IF iState >= 10 AND iState < 100 THEN 
	THIS^.M_0ReadActConfig();
ELSIF iState >= 1000 AND iState < 1100 THEN
//	act11_DownloadDriveFirmware();				// Execute this Action in a different Task
 	iState := 100; 
ELSIF iState >= 100 AND iState < 200 THEN
	THIS^.M_1ConfigAxes();
ELSIF iState >= 200 AND iState < 300 THEN
	THIS^.M_2ConfigSercosIO();
ELSIF iState >= 300 AND iState < 400 THEN
	THIS^.M_3ConfigInlineIO();	
ELSIF iState >= 400 AND iState < 500 THEN
	THIS^.M_4ConfigProfibsIO();
ELSIF iState >= 500 AND iState < 600 THEN
	iState := 800;
ELSIF iState >= 800 AND iState < 900 THEN
	THIS^.M_8WriteConfig();
ELSIF iState >= 900 AND iState < 1000 THEN
	THIS^.M_9ErrorDone();
END_IF
END_METHOD

METHOD PRIVATE M_GetSafetyType : STRING(2)
VAR_INPUT
	///Temp string to prepare elements;
	apsTypeCodeElements: ARRAY[1..20] OF POINTER TO STRING(255);
	bSecondDoubleAxis: BOOL := FALSE;
END_VAR
IF (LEFT (apsTypeCodeElements[1]^,5) = 'CSH01') THEN

	M_GetSafetyType := apsTypeCodeElements[6]^;
	
ELSIF	(LEFT (apsTypeCodeElements[1]^,5) = 'CDB01') THEN

	M_GetSafetyType := apsTypeCodeElements[7]^;
	
ELSIF	(LEFT (apsTypeCodeElements[1]^,5) = 'CSE02') 
OR	(LEFT (apsTypeCodeElements[1]^,5) = 'CSB02')
OR	(LEFT (apsTypeCodeElements[1]^,5) = 'CSH02') 
OR	(LEFT (apsTypeCodeElements[1]^,5) = 'CSB01') 
OR	(LEFT (apsTypeCodeElements[1]^,5) = 'KMC02') THEN		(* 2019-03-21 Bär: Typ 'KMC02' im Rahmen der RDK90 (Mi-Antriebe) hinzugefügt *)

	M_GetSafetyType := apsTypeCodeElements[5]^;
	
ELSIF	(LEFT (apsTypeCodeElements[1]^,5) = 'CDB02') THEN

	IF NOT bSecondDoubleAxis THEN
		M_GetSafetyType := apsTypeCodeElements[6]^;
	ELSE	
		M_GetSafetyType := apsTypeCodeElements[7]^;
	END_IF
	
ELSIF	(LEFT (apsTypeCodeElements[1]^,5) = 'HCS01') THEN

	M_GetSafetyType := apsTypeCodeElements[9]^;
	
ELSIF	(LEFT (apsTypeCodeElements[1]^,5) = 'KSM02') 
OR	(LEFT (apsTypeCodeElements[1]^,5) = 'KMS02')THEN

	M_GetSafetyType := apsTypeCodeElements[7]^;
	
END_IF
END_METHOD

///FUNCTION FUN_GetSercosAdress
///
///General Header
///----------------------------------------------------------------------------------------------
///Short description      : extract sercos adress for double axis config
///Version                : 13.0.0
///Author                 : Jörg Schneider
///Date                   : 13-07-12 15:46:38
///Company                : DC-IA
///Target                 : MLC 13 ff
///----------------------------------------------------------------------------------------------
METHOD PRIVATE M_GetSercosAdress : INT
VAR_INPUT
	/// Pointer to String Element of C-0-0479 e.g. 'V3|34' 
	pbToElement: POINTER TO BYTE;
	/// First or second Adress of doubleAxis
	iNoOfAddress: INT;
END_VAR
VAR
	sTemp: STRING := '';
	sTemp2: STRING := '';
	pbTemp: POINTER TO BYTE;
	pbTemp2: POINTER TO BYTE;
	psStringTemp: POINTER TO STRING(1);
	bTemp: BYTE;
	iDigit1: INT;
	iDigit2: INT;
END_VAR
// copy first sign to stTemp 				
pbTemp := pbToElement+1;	
psStringTemp := pbTemp;					
sTemp := psStringTemp^;
bTemp := pbTemp^;
		
sTemp2 := '';		
pbTemp2 := ADR (sTemp2);



// Do until '|' or end of string appears				
IF NOT (sTemp = '') 			// End of String
AND NOT (bTemp = 124) THEN		// Or '|' character
	pbTemp2^:= pbTemp^;

	iDigit1 := STRING_TO_INT(sTemp);
	iDigit2 := 0;
	
	pbTemp := pbTemp + 1;
	pbTemp2 := pbTemp2 + 1;
	psStringTemp := pbTemp;
	sTemp := psStringTemp^;
	bTemp := pbTemp^;

	
END_IF	

IF NOT (sTemp = '') 
AND NOT (bTemp = 124) THEN
	pbTemp2^:= pbTemp^;
	
	iDigit1 := iDigit1 *10;
	iDigit2 := STRING_TO_INT(sTemp);
		
	pbTemp := pbTemp + 1;
	pbTemp2 := pbTemp2 + 1;
	psStringTemp := pbTemp;
	sTemp := psStringTemp^;
	bTemp := pbTemp^;
	
END_IF	


IF iNoOfAddress = 2 THEN 
	//Reset Temp variable
	sTemp2 := '';		
	pbTemp2 := ADR (sTemp2);
	pbTemp := pbTemp + 1;
	psStringTemp := pbTemp;
	sTemp := psStringTemp^;


	IF NOT (sTemp = '')  THEN
		pbTemp2^:= pbTemp^;
					
		iDigit1 := STRING_TO_INT(sTemp);
		iDigit2 := 0;
				
		pbTemp := pbTemp + 1;
		pbTemp2 := pbTemp2 + 1;
		psStringTemp := pbTemp;
		sTemp := psStringTemp^;
		bTemp := pbTemp^;
	
	END_IF	
	
	IF NOT (sTemp = '')  THEN
		pbTemp2^:= pbTemp^;
		
		iDigit1 := iDigit1 *10;
		iDigit2 := STRING_TO_INT(sTemp);
		
		pbTemp := pbTemp + 1;
		pbTemp2 := pbTemp2 + 1;
		psStringTemp := pbTemp;
		sTemp := psStringTemp^;
		bTemp := pbTemp^;
		
		
	END_IF	

END_IF


M_GetSercosAdress := iDigit1 + iDigit2;
END_METHOD

METHOD PRIVATE M_S20TypeToString : STRING
VAR_INPUT
	eS20Type: E_S20Type;
END_VAR
CASE eS20Type OF
	
	E_S20Type.S20_UNDEFINED				:	M_S20TypeToString :=  'undefinded'				;
	E_S20Type.S20_S3_BK_PLUS				:	M_S20TypeToString :=  'S20-S3-BK+'	            ;
	E_S20Type.S20_DI_16_4     		   	:	M_S20TypeToString :=  'S20-DI-16/4'	            ;
	E_S20Type.S20_DO_16_3          		:	M_S20TypeToString :=  'S20-DO-16/3'	            ;
	E_S20Type.S20_DI_32_1          		:	M_S20TypeToString :=  'S20-DI-32/1'	            ;
	E_S20Type.S20_DO_32_1          		:	M_S20TypeToString :=  'S20-DO-32/1'	            ;
	E_S20Type.S20_DO_8_2_2A        		:	M_S20TypeToString :=  'S20-DO-8/2-2A'            ;
	E_S20Type.S20_DI_16_1          		:	M_S20TypeToString :=  'S20-DI-16/1'	            ;
	E_S20Type.S20_DO_16_1          		:	M_S20TypeToString :=  'S20-DO-16/1'	            ;
	E_S20Type.S20_AI_8             		:	M_S20TypeToString :=  'S20-AI-8'		            ;
	E_S20Type.S20_AI_8_RTD         		:	M_S20TypeToString :=  'S20-AI-8-RTD'	            ;
	E_S20Type.S20_AI_8_UTH         		:	M_S20TypeToString :=  'S20-AI-8-UTH'	            ;
	E_S20Type.S20_AO_8             		:	M_S20TypeToString :=  'S20-AO-8'		            ;
	E_S20Type.S20_CNT_INC_2_2      		:	M_S20TypeToString :=  'S20-CNT-INC-2/2'	        ;
	E_S20Type.S20_SSI_AO_1_1       		:	M_S20TypeToString :=  'S20-SSI-AO-1/1'	        ;
	E_S20Type.Placeholder_1          		:	M_S20TypeToString :=  'Test_ChM'			        ;
	E_S20Type.Placeholder_2 		     	:	M_S20TypeToString :=  'Test_ChM'			        ;
	E_S20Type.Placeholder_3          		:	M_S20TypeToString :=  'Test_ChM'			        ;
	E_S20Type.S20_AI_4_I           		:	M_S20TypeToString :=  'S20-AI-4-I'		        ;
	E_S20Type.S20_AI_4_U           		:	M_S20TypeToString :=  'S20-AI-4-U'		        ;
	E_S20Type.S20_DI_64_1    			   	:	M_S20TypeToString :=  'S20-DI-64/1'		        ;
	E_S20Type.S20_DI_16_1_HS     	 		:	M_S20TypeToString :=  'S20-DI-16/1-HS'	        ;
	E_S20Type.S20_AI_4_RTD         		:	M_S20TypeToString :=  'S20-AI-4-RTD'		        ;
	E_S20Type.S20_RS_UNI           		:	M_S20TypeToString :=  'S20-RS-UNI'		        ;
	E_S20Type.S20_DIDO_8_1         		:	M_S20TypeToString :=  'S20-DIDO-8/1'		        ;
	E_S20Type.S20_AO_4             		:	M_S20TypeToString :=  'S20-AO-4'                 ;
	E_S20Type.S20_AI_4_UTH         		:	M_S20TypeToString :=  'S20-AI-4-UTH'		        ;
	E_S20Type.S20_SSDI_8_4               	:	M_S20TypeToString:=  'SSDI-8/4'			        ;
	E_S20Type.S20_SSDO_8_3               	:	M_S20TypeToString:=  'SSDO-8/3'			        ;
	E_S20Type.S20_AI6_AO2_SSI2     		:	M_S20TypeToString:=  'S20-AI6-AO2-SSI2'	        ;
	E_S20Type.S20_INC_2            		:	M_S20TypeToString:=  'S20-INC-2'		        ;
	E_S20Type.S20_AIAO_2           		:	M_S20TypeToString:=  'S20-AIAO-2'		        ;
	E_S20Type.S20_DO_64_1          		:	M_S20TypeToString:=  'S20-DO-64/1'				;	
	E_S20Type.S20_DOR_4_2_220_AC   		:	M_S20TypeToString:=  'S20-DOR-4/2-220-AC'		;	
	E_S20Type.S20_DI_16_4_DO_8_3_HS		:	M_S20TypeToString:=  'S20-DI-16/4-DO-8/3-HS'	;	
															  	
END_CASE
END_METHOD

METHOD PRIVATE M_TypeCodeIsRexrothIO : BOOL
VAR_INPUT
	sTypeCode: STRING;
END_VAR

IF sTypeCode = 'L05R911172531' THEN			// S20-S3-BK
	M_TypeCodeIsRexrothIO := TRUE;
ELSIF 	sTypeCode = 'L05R911173318' THEN		// S20-S3-BK+
	M_TypeCodeIsRexrothIO := TRUE;
ELSIF 	sTypeCode = 'L05R911170875' THEN		// R-IL S3 BK DI8 DO4-PAC
	M_TypeCodeIsRexrothIO := TRUE;	
ELSIF 	sTypeCode = 'L05R911170874' THEN		// R-ILB S3 AI4 AO2
	M_TypeCodeIsRexrothIO := TRUE;
ELSIF 	sTypeCode = 'L05R911171676' THEN		// R-ILB S3 AI6 AO4/F
	M_TypeCodeIsRexrothIO := TRUE;
ELSIF 	sTypeCode = 'L05R911171949' THEN		// R-ILB S3 AI12 AO4 SSI-IN4
	M_TypeCodeIsRexrothIO := TRUE;
ELSIF 	sTypeCode = 'L05R911170826' THEN		// R-ILB S3 24 DI16 DIO16
	M_TypeCodeIsRexrothIO := TRUE;
ELSIF 	sTypeCode = 'L05R911171675' THEN		// R-ILB S3 24 DI16 DIO16/F
	M_TypeCodeIsRexrothIO := TRUE;
ELSIF 	sTypeCode = 'L05R911172899' THEN		// S67-S3-BK-DI8-M8
	M_TypeCodeIsRexrothIO := TRUE;

ELSE 	
	M_TypeCodeIsRexrothIO := FALSE;
END_IF
END_METHOD

END_FUNCTION_BLOCK

// GeneralFunctionBlocks/ActivateDevices/ITF_ActivateDevices
INTERFACE ITF_ActivateDevices

METHOD M_Execute
END_METHOD

END_INTERFACE

// GeneralFunctionBlocks/ChangeNextDiagDelay/FB_ChangeNextDiagDelay
{attribute 'qualified_only' := ''}
{attribute 'namespace' := 'ILGStdLib.FunctionBlocks'}
FUNCTION_BLOCK FB_ChangeNextDiagDelay
VAR_INPUT
	/// start procedure
	IN_bExecute: BOOL;
	/// Delay Time in ms
	IN_diDiagDelayTime: DINT;
END_VAR
VAR_OUTPUT
	/// Done
	OUT_bDone: BOOL;
	/// Active
	OUT_bActive: BOOL;
	/// error	
	OUT_bError: BOOL;
	/// internat state when error occured
	OUT_iErrorState: INT;
END_VAR
VAR CONSTANT
	/// max no of directory entries
	iMaxDirEntry: INT := 400;
END_VAR
VAR
	bExecuteOld: BOOL;
	istate: INT;
	iLength: INT;
	i: INT;
	j: INT;
	iEOF: INT;
	hCfg: ITF_FILEASYNC;
	sBuffer: STRING(7000);
	udiReadBytes: UDINT;
	udiFileSize: UDINT;
	sLineFeed: STRING(1);
	sTemp: STRING;
	sTemp2: STRING;
	sSearch: STRING;
	diResult: DINT;
	astSplit: ST_Split;
	asStringFile: ARRAY[1..iMaxDirEntry] OF STRING;
	psFileName : POINTER TO STRING;
	psNewFileName : POINTER TO STRING;
	fb_ILFileDeleteAsync: IL_FileDeleteAsync;
	fb_ILFileOpenAsync: IL_FileAsync;
	fb_ILFileReadAsync: IL_FileReadAsync;	
	fb_ILFileGetSizeAsync: IL_FileGetSizeAsync;
	fb_ILFileRenameAsync: IL_FileRenameAsync;
	fb_ILFileWriteAsync: IL_FileWriteAsync;
END_VAR


IF IN_bExecute AND NOT bExecuteOld THEN
	bExecuteOld := TRUE;
	OUT_bActive := TRUE;
	OUT_bDone := FALSE;
	OUT_bError := FALSE;
	iState := 40;
END_IF	

IF NOT IN_bExecute AND bExecuteOld 
	AND (OUT_bDone OR OUT_bError) THEN
	bExecuteOld := FALSE;
	OUT_bActive := FALSE;
	OUT_bDone := FALSE;
	OUT_bError := FALSE;
	iState := 0;
END_IF	


CASE istate OF

40: // Größe ermitteln
	psFileName^:= '/ata0a/ProjectData/PLC/DevicePLcAdd.cfg';
	OUT_iErrorState := iState;
	fb_ILFileGetSizeAsync(
		Execute:=TRUE , 
		FileName:= psFileName,			(* 2016-10 gt: IW13: '/ata0a/DevicePLcAdd.cfg' --> IW14: '/ata0a/ProjectData/PLC/DevicePLcAdd.cfg' *) (* 2017-01-26 gt: relevant für IW14 *)
		Done=> ,		
		Active=> ,
		Error=> ,
 		ErrorId=> ,
		ErrorIdent=> , 
		FileSize=> udiFileSize);

	IF fb_ILFileGetSizeAsync.Done THEN
		fb_ILFileGetSizeAsync(
			Execute:= FALSE);
		iState :=50;
	END_IF
	// Error	
	IF fb_ILFileGetSizeAsync.Error THEN
		fb_ILFileGetSizeAsync(
			Execute:= FALSE);
		iState :=999;
	END_IF
			
50:	// DevicePlcAdd.cfg öffnen
	psFileName^:= '/ata0a/ProjectData/PLC/DevicePLcAdd.cfg';
	OUT_iErrorState := iState;		
	fb_ILFileOpenAsync(
		Enable:= TRUE, 
		FileName:=psFileName,		(* 2016-10 gt: IW13: '/ata0a/DevicePLcAdd.cfg' --> IW14: '/ata0a/ProjectData/PLC/DevicePLcAdd.cfg' *) (* 2017-01-26 gt: relevant für IW14 *)
		Mode:=  AM_READ,
		InOperation=> , 
		Active=> ,
		Shutdown=> , 		 
		Error=> , 
		ErrorId=> ,
		ErrorIdent=> , 
		FileHandle=> hCfg);

	IF fb_ILFileOpenAsync.InOperation THEN		
		sBuffer := '';	
		iState :=60;
	END_IF

	// Error	
	IF fb_ILFileOpenAsync.Error THEN
		fb_ILFileOpenAsync(
			Enable:= FALSE);
		iState :=999;
	END_IF
		
60:	// DevicePlcAdd.cfg lesen
	OUT_iErrorState := iState;
	fb_ILFileReadAsync(
		Execute:= TRUE,
		BufferAddr:= ADR(sBuffer),
 		BufferSize:= udiFileSize, 
		FileHandle:= hCfg,  
		Done=> , 
		Active=> , 
		Error=> , 
		ErrorId=> ,
		ErrorIdent=> , 
		BytesRead=> udiReadBytes );

	IF fb_ILFileReadAsync.Done THEN
		fb_ILFileReadAsync(
			Execute:= FALSE);
		iState := 70;
	END_IF

	// Error	
	IF fb_ILFileReadAsync.Error THEN
		fb_ILFileReadAsync(
			Execute:= FALSE);
		iState :=999;
	END_IF
	
70: // Datei schließen
	OUT_iErrorState := iState;
	fb_ILFileOpenAsync(
		Enable:= FALSE); 

	IF (fb_ILFileOpenAsync.InOperation = FALSE) THEN
		iState :=80;
	END_IF

	// Error	
	IF fb_ILFileOpenAsync.Error THEN
		iState :=999;
	END_IF
	
	(* Auskommentiert, da strSplit strLen usw. noch fehlen
80: // Datei in Array of String kopieren und Formatzeichen löschen
	OUT_iErrorState := iState;
	strSplit(ADR(sBuffer),13 ,0,FALSE,ADR(astSplit));
	sLineFeed := CHR(10);
	
	FOR i := 1 TO iMaxDirEntry DO 
		IF astSplit.arWords[i]^ = astSplit.arWords[iMaxDirEntry]^ THEN 
			iEOF := i ;		
			i := iMaxDirEntry;
		END_IF
		asStringFile[i] := DEL_CHARS(astSplit.arWords[i]^, sLineFeed);
	END_FOR
	
	// letzte Zeile löschen
	asStringFile[iEOF-1] := ''; 
	iEOF	:= iEOF-2;
	
	iState := 90;	

90:	// Sektion im File suchen
	OUT_iErrorState := iState;
	sSearch := '[NetX_Device]';  
	iLength :=	strLen(ADR(sSearch));
	FOR i := 1 TO iEOF DO
		sTemp := '';
		IF strLen(ADR(asStringFile[i])) >= iLength THEN									// Text länger als strSearch
			
			IF (asStringFile[i] = sSearch) THEN					// Text enthält '[NetX_Device]'
				sSearch := 'NetxDiagDelayTime=';
				iLength :=	strLen(ADR(sSearch));
				strNCopy(ADR(sTemp), (INT_TO_UINT(iLength)+2), ADR(asStringFile[i+1]), iLength);		(* 2014-11-14 gt: INT_TO_UINT() hinzu, wegen Warnung *)
				
				IF NOT (sTemp = sSearch) THEN					// Text enthält noch nicht 'NetxDiagDelayTime='
					FOR j:= iEOF TO i+1 BY -1 DO					// dann alle Zeilen um eins nach unten verschieben
						asStringFile[j+1] := asStringFile[j];	
					END_FOR
			
					asStringFile[i+1] := 'NetxDiagDelayTime=';		// Zeile inzufügen.
					sTemp := DINT_TO_STRING(IN_diDiagDelayTime);
					strConcat(ADR(asStringFile[i+1]), SIZEOF(asStringFile[i+1]), ADR(sTemp));
				ELSE																	// Text enthält 'NetxDiagDelayTime='
					sTemp := 'NetxDiagDelayTime=';		
					sTemp2 := DINT_TO_STRING(IN_diDiagDelayTime);
					strConcat(ADR(sTemp), SIZEOF(sTemp), ADR(sTemp2));
					IF sTemp = asStringFile[i+1] THEN  // Vergleichen, ob Wert stimmt 
						i := iEOF+1;
						iState := 250;  									// --> Done
						RETURN;
					ELSE
						asStringFile[i+1] := sTemp; 		// Zeile neu schreiben
					END_IF		
				END_IF
				i := iEOF+1; // End FOR Loop
			END_IF
		END_IF	
	END_FOR	
	
	iState := 110;
	*)
110: // DevicePlcAdd.new neu anlegen und zum schreiben öffnen
	psFileName^:= '/ata0a/ProjectData/PLC/DevicePLcAdd.new';
	OUT_iErrorState := iState;
	// hCfg := SysFileStreamFOpenV3('/ata0a/ProjectData/PLC/DevicePLcAdd.new', 'w');		(* 2016-10 gt: IW13: ('/ata0a/DevicePLcAdd.new', 'w') --> IW14: ('/ata0a/ProjectData/PLC/DevicePLcAdd.new', 'w') *)	(* 2017-01-26 gt: relevant für IW14 *)
	fb_ILFileOpenAsync(
		Enable:= TRUE, 
		FileName:=psFileName,		(* 2016-10 gt: IW13: '/ata0a/DevicePLcAdd.cfg' --> IW14: '/ata0a/ProjectData/PLC/DevicePLcAdd.cfg' *) (* 2017-01-26 gt: relevant für IW14 *)
		Mode:=  AM_WRITE,
		InOperation=> , 
		Active=> ,
		Shutdown=> , 		 
		Error=> , 
		ErrorId=> ,
		ErrorIdent=> , 
		FileHandle=> hCfg);

	IF fb_ILFileOpenAsync.InOperation THEN					
		iState :=120;
		j := 0;
	END_IF

	// Error	
	IF fb_ILFileOpenAsync.Error THEN
		fb_ILFileOpenAsync(
			Enable:= FALSE);
		iState :=999;
	END_IF
		
	
120:
	OUT_iErrorState := iState;
	FOR i := j+1 TO iEOF DO
		diResult := FUN_WriteLnString(hCfg, asStringFile[i]);
(*		IF i >= j+10 THEN
			j := i;
			RETURN;
		END_IF  	*)
	END_FOR
	iState :=130;

130:
	OUT_iErrorState := iState;
	
	fb_ILFileOpenAsync(
		Enable:= FALSE);
	iState :=140;

140: // alte Datei umbenennen
	psFileName^ := '/ata0a/ProjectData/PLC/DevicePLcAdd.cfg';
	psNewFileName^ := '/ata0a/ProjectData/PLC/DevicePLcAdd.old'; 
	OUT_iErrorState := iState;
	fb_ILFileRenameAsync(
		Execute:= TRUE, 
		OldName:= psFileName, 		(* 2016-10 gt: IW13: '/ata0a/DevicePLcAdd.cfg' --> IW14: '/ata0a/ProjectData/PLC/DevicePLcAdd.cfg' *)	(* 2017-01-26 gt: relevant für IW14 *)
		NewName:= psNewFileName, 		(* 2016-10 gt: IW13: '/ata0a/DevicePLcAdd.old' --> IW14: '/ata0a/ProjectData/PLC/DevicePLcAdd.old' *)	(* 2017-01-26 gt: relevant für IW14 *)
		Done=> , 
		Active=> , 
		Error=> , 
		ErrorId=> ,
		ErrorIdent=>);
	
	IF fb_ILFileRenameAsync.Done THEN
		fb_ILFileRenameAsync(
			Execute:= FALSE);
		iState :=150;
	END_IF

		// Error	
	IF fb_ILFileRenameAsync.Error THEN
		fb_ILFileRenameAsync(
			Execute:= FALSE);
		iState :=999;
	END_IF

150: // neue Datei umbenennen
	psFileName^ := '/ata0a/ProjectData/PLC/DevicePLcAdd.new';
	psNewFileName^ := '/ata0a/ProjectData/PLC/DevicePLcAdd.cfg';
	OUT_iErrorState := iState;	
	fb_ILFileRenameAsync(
		Execute:= TRUE, 
		OldName:= psFileName, 		(* 2016-10 gt: IW13: '/ata0a/DevicePLcAdd.new' --> IW14: '/ata0a/ProjectData/PLC/DevicePLcAdd.new' *)	(* 2017-01-26 gt: relevant für IW14 *)
		NewName:= psNewFileName,		(* 2016-10 gt: IW13: '/ata0a/DevicePLcAdd.cfg' --> IW14: '/ata0a/ProjectData/PLC/DevicePLcAdd.cfg' *) (* 2017-01-26 gt: relevant für IW14 *)
		Done=> , 
		Active=> , 
		Error=> , 
		ErrorId=> ,
		ErrorIdent=> );
	
	IF fb_ILFileRenameAsync.Done THEN
		fb_ILFileRenameAsync(
			Execute:= FALSE);
		iState :=160;
	END_IF

	// Error	
	IF fb_ILFileRenameAsync.Error THEN
		fb_ILFileRenameAsync(
			Execute:= FALSE);
		iState :=999;
	END_IF
	
160: // alte Datei löschen
	psFileName^ := '/ata0a/ProjectData/PLC/DevicePLcAdd.old';
	OUT_iErrorState := iState;
	fb_ILFileDeleteAsync(
		Execute:= TRUE, 
		FileName:= psFileName, 		(* 2016-10 gt: IW13: '/ata0a/DevicePLcAdd.old' --> IW14: '/ata0a/ProjectData/PLC/DevicePLcAdd.old' *)	(* 2017-01-26 gt: relevant für IW14 *)
		Done=> , 
		Active=> , 
		Error=> , 
		ErrorId=> ,
		ErrorIdent=> );
	
	IF fb_ILFileDeleteAsync.Done THEN
		fb_ILFileDeleteAsync(
			Execute:= FALSE);
		i := 0;
		iState :=250;
	END_IF

	// Error	
	IF fb_ILFileDeleteAsync.Error THEN
		fb_ILFileDeleteAsync(
			Execute:= FALSE);
		iState :=999;
	END_IF

250:  // Done
	OUT_iErrorState := 0;
	OUT_bDone := TRUE;
	OUT_bActive := FALSE;	
	OUT_bError := FALSE;

999: // ERROR 
	OUT_bDone := FALSE;
	OUT_bActive := FALSE;	
	OUT_bError := TRUE;
	
END_CASE

END_FUNCTION_BLOCK

// GeneralFunctions/Convert/F_byWordToLeftByte
{attribute 'qualified_only' := ''}
{attribute 'namespace' := 'ILGStdLib.Functions.Convert'}
FUNCTION F_byWordToLeftByte : BYTE
VAR_INPUT
	/// Zu spaltendes Wort 
	In_wInput: WORD;
END_VAR
VAR
	pwWord: POINTER TO WORD;
	wTEMP: WORD;
END_VAR

pwWord:= ADR(In_wInput);
pwWord:= (pwWord+1);
wTEMP:= pwWord^;
F_byWordToLeftByte:= WORD_TO_BYTE(wTEMP);

END_FUNCTION

// GeneralFunctions/Convert/F_DwordToStrH5
{attribute 'qualified_only' := ''}
{attribute 'namespace' := 'ILGStdLib.Functions.Convert'}
FUNCTION F_DwordToStrH5 : STRING(5)
VAR_INPUT
	In_dwInput: DWORD;
END_VAR
VAR
	i: INT;
	byTemp: BYTE;
	pbyOut: POINTER TO BYTE;
END_VAR

//read output adress
pbyOut := ADR(F_DwordToStrH5) + 5;
// write last byte of String 
pbyOut^:= 0;

// write the 5 hex characters backwards 
FOR i := 1 TO 5 DO
	//decrement pointer
	pbyOut := pbyOut - 1;
	// read the lowest value
	byTemp := DWORD_TO_BYTE(In_dwInput AND 16#0000F);
	// convert value to hex 
	IF (byTemp <= 9) THEN 
		byTemp := byTemp + 48; 
	ELSE 
		byTemp := byTemp + 55; 
	END_IF
	// write value to string
	pbyOut^ := byTemp;
	//shift input for next hex digit
	In_dwInput := SHR(In_dwInput,4);
END_FOR

END_FUNCTION

// GeneralFunctions/Convert/F_DwordToStrH8
{attribute 'qualified_only' := ''}
{attribute 'namespace' := 'ILGStdLib.Functions.Convert'}
FUNCTION F_DwordToStrH8 : STRING(8)
VAR_INPUT
	In_dwInput: DWORD;
END_VAR
VAR
	i: INT;
	byTemp: BYTE;
	pbyOut: POINTER TO BYTE;
END_VAR

//read output adress
pbyOut := ADR(F_DwordToStrH8) + 8;
// write last byte of String 
pbyOut^:= 0;

// write the 8 hex characters backwards 
FOR i := 1 TO 8 DO
	//decrement pointer
	pbyOut := pbyOut - 1;
	// read the lowest value
	byTemp := DWORD_TO_BYTE(In_dwInput AND 16#0000000F);
	// convert value to hex 
	IF (byTemp <= 9) THEN 
		byTemp := byTemp + 48; 
	ELSE 
		byTemp := byTemp + 55; 
	END_IF
	// write value to string
	pbyOut^ := byTemp;
	//shift input for next hex digit
	In_dwInput := SHR(In_dwInput,4);
END_FOR

END_FUNCTION

// GeneralFunctions/Convert/F_dwSwapDWordWord
{attribute 'qualified_only' := ''}
{attribute 'namespace' := 'ILGStdLib.Functions.Convert'}
FUNCTION F_dwSwapDWordWord : DWORD
VAR_INPUT
	In_dwInput: DWORD;
END_VAR
VAR
	pwWordIn: POINTER TO ARRAY[1..2] OF WORD;
	pwWordOut: POINTER TO ARRAY[1..2] OF WORD;
	dwOutput: DWORD;
END_VAR


pwWordIn := ADR(In_dwInput);
pwWordOut := ADR(dwOutput);

pwWordOut^[1]	:=	pwWordIn^[2] ;
pwWordOut^[2]	:=	pwWordIn^[1] ;

F_dwSwapDWordWord := dwOutput;

END_FUNCTION

// GeneralFunctions/Convert/F_iAnalogOutput4To20mA
{attribute 'qualified_only' := ''}
{attribute 'namespace' := 'ILGStdLib.Functions.Convert'}
FUNCTION F_iAnalogOutput4To20mA : INT
VAR_INPUT
	/// x;  Wert zur Wandlung für die Analogausgabe 
	In_rValueToConvert: REAL;
	/// y1; Dezimalwert bei 4mA an Analogausgabe: z.B.      0 
	In_iDecimal4mA: INT;
	/// y2; Dezimalwert bei 20mA an Analogausgabe: z.B. 30000 
	In_iDecimal20mA: INT;
	/// x1; Minimalwert für die Wandlung bei 4mA: z.B. Position    0mm 
	In_rConversionMinValue4mA: REAL;
	/// x2; Maximalwert für die Wandlung bei 20mA: z.B. Position 140mm 
	In_rConversionMaxValue20mA: REAL;
END_VAR
VAR
	/// Differenz zwischen Dezimalwert von 20mA und 4mA 
	rDecimalDifference: REAL;
	/// Differenz zwischen Minimalwert und Maximalwert der Wandlung 
	rConversionDifference: REAL;
END_VAR

(* Geradengleichung: y = y1 + (y2-y1)/(x2-x1) * (x-x1) *)

(* Differenz zwischen Dezimalwert von 20mA und 4mA *)
rDecimalDifference := INT_TO_REAL(In_iDecimal20mA - In_iDecimal4mA);					(* entspricht (y2-y1) *)

(* Differenz zwischen Minimalwert und Maximalwert der Wandlung *)
rConversionDifference := In_rConversionMaxValue20mA - In_rConversionMinValue4mA;	(* entspricht (x2-x1) *)


(* Geradengleichung:  y  =                          y1              + (y2-y1)              / (x2-x1)               * (x-x1) *)
F_iAnalogOutput4To20mA := REAL_TO_INT(INT_TO_REAL(In_iDecimal4mA) + (rDecimalDifference) / (rConversionDifference) * (In_rValueToConvert - In_rConversionMinValue4mA));

END_FUNCTION

// GeneralFunctions/Convert/F_rAnalogInput0To10V
{attribute 'qualified_only' := ''}
{attribute 'namespace' := 'ILGStdLib.Functions.Convert'}
FUNCTION F_rAnalogInput0To10V : REAL
VAR_INPUT
	/// x;  Wert von Analogeingabe 
	In_iValueToConvert: INT;
	/// x1; [Digit] Dezimalwert bei 0V von Analogeingabe: z.B.      0 
	In_iDecimal0V: INT;
	/// x2; [Digit] Dezimalwert bei 10V von Analogeingabe: z.B. 10000 
	In_iDecimal10V: INT;
	/// y1; Minimalwert der Wandlung bei 0V: z.B. Position    0mm 
	In_rConversionMinValue0V: REAL;
	/// y2; Maximalwert der Wandlung bei 10V: z.B. Position  10mm 
	In_rConversionMaxValue10V: REAL;
END_VAR
VAR
	/// Differenz zwischen Dezimalwert von 10V und 0V 
	rDecimalDifference: REAL;
	/// Differenz zwischen Minimalwert und Maximalwert der Wandlung 
	rConversionDifference: REAL;
END_VAR

(* Geradengleichung: y = y1 + (y2-y1)/(x2-x1) * (x-x1) *)

(* Differenz zwischen Dezimalwert von 10V und 0V *)
rDecimalDifference := INT_TO_REAL(In_iDecimal10V - In_iDecimal0V);					(* entspricht (x2-x1) *)

(* Differenz zwischen Minimalwert und Maximalwert der Wandlung *)
rConversionDifference := In_rConversionMaxValue10V - In_rConversionMinValue0V;		(* entspricht (y2-y1) *)


(* Geradengleichung:  y  =                          y1  + (y2-y1)               / (x2-x1)              * (x-x1) *)
(* 2013-12-19 Carle: geändert STAL 90 *)
//rWert_Analogeingabe_out := (INT_TO_REAL(iDezimal_0V_in) + (rWandlung_Differenz) / (rDezimal_Differenz) * INT_TO_REAL(iWert_zur_Wandlung_in - iDezimal_0V_in));
F_rAnalogInput0To10V := (In_rConversionMinValue0V + (rConversionDifference) / (rDecimalDifference) * INT_TO_REAL(In_iValueToConvert - In_iDecimal0V));

END_FUNCTION

// GeneralFunctions/Convert/F_rSwapReal
{attribute 'qualified_only' := ''}
{attribute 'namespace' := 'ILGStdLib.Functions.Convert'}
FUNCTION F_rSwapReal : REAL
VAR_INPUT
	In_rInput: REAL;
END_VAR
VAR
	pDword: POINTER TO DWORD;
	pReal: POINTER TO REAL;
	dwOutput: DWORD;
END_VAR

pDword := ADR(In_rInput);
dwOutput := IL_SwapDWord(pDword^);
pReal := ADR(dwOutput);
F_rSwapReal := pReal^;

END_FUNCTION

// GeneralFunctions/Convert/F_rSwapRealWord
{attribute 'qualified_only' := ''}
{attribute 'namespace' := 'ILGStdLib.Functions.Convert'}
FUNCTION F_rSwapRealWord : REAL
VAR_INPUT
	In_rInput: REAL;
END_VAR
VAR
	pwWordIn: POINTER TO ARRAY[1..2] OF WORD;
	pwWordOut: POINTER TO ARRAY[1..2] OF WORD;
	rOutput: REAL;
END_VAR


pwWordIn := ADR(In_rInput);
pwWordOut := ADR(rOutput);

pwWordOut^[1]	:=	pwWordIn^[2] ;
pwWordOut^[2]	:=	pwWordIn^[1] ;

F_rSwapRealWord := rOutput;

END_FUNCTION

// GeneralFunctions/Convert/F_Tad
FUNCTION F_Tad
(* High-/ LoByte der Übergabevariable tauschen und an gleicher Stelle speichern*)
VAR_INPUT
	pdwValue: POINTER TO DWORD;
END_VAR
VAR
END_VAR

pdwValue^ := IL_SwapDWord(pdwValue^);	(* High-/ LoByte der Übergabevariable tauschen und an gleicher Stelle speichern*)

END_FUNCTION

// GeneralFunctions/Convert/F_WordToStrH
{attribute 'qualified_only' := ''}
{attribute 'namespace' := 'ILGStdLib.Functions.Convert'}
FUNCTION F_WordToStrH : STRING(4)
VAR_INPUT
	In_dwInput: DWORD;
END_VAR
VAR
	i: INT;
	byTemp: BYTE;
	pbyOut: POINTER TO BYTE;
END_VAR

(* read output adress to pointer *)
pbyOut := ADR(F_WordToStrH) + 4;
(* wirte the closing byte for the string *)
pbyOut^:= 0;

(* write the 8 hex characters backwards *)
FOR i := 1 TO 4 DO;
	(* decrement the pointer *)
	pbyOut := pbyOut - 1;
	(* read the lowest order hex value *)
	byTemp := DWORD_TO_BYTE(In_dwInput AND 16#0000000F);
	(* convert value to hex character *)
	IF byTemp <= 9 THEN byTemp := byTemp + 48; ELSE byTemp := byTemp + 55; END_IF;
	(* write character to output string *)
	pbyOut^ := byTemp;
	(* shift in for nect hex character *)
	In_dwInput := SHR(In_dwInput,4);
END_FOR;

END_FUNCTION

// GeneralFunctions/ILG_Functions/F_bCamDiscCalculation
{attribute 'qualified_only'}
{attribute 'namespace' := 'ILGStdLib.Functions.ILG_Functions' }
FUNCTION F_bCamDiscCalculation : BOOL
VAR_INPUT
	In_padiCam     	: POINTER TO ARRAY [1..1024] OF DINT;
	In_iLoopCount  	: INT;
	In_iStepNo     	: INT;
	In_iAxisNo     	: INT;
	In_iCamNo      	: INT;
	In_lrMasterSeg	: LREAL;
	In_lrHubG     	: LREAL;
	In_lrHubRG   	: LREAL;
	paaarServoAxes	: POINTER TO T_ServoAxesArray;	(* Übergabe pointer globales array Array_Servoachsen *)
END_VAR
VAR_IN_OUT
	paarCamTable	: POINTER TO T_CamTable;		(* Übergabe pointer globales array arKurventabelle *)
	paarTabArray		: POINTER TO T_Tables;			(* Übergabe pointer globales array Tab_Array *)
END_VAR
VAR
	iBewegGesetzSeg :INT;
	
END_VAR

iBewegGesetzSeg:= REAL_TO_INT(paaarServoAxes^[In_iAxisNo,In_iStepNo,1]);

IF In_lrMasterSeg > 0.0 THEN
	paarCamTable^[In_iCamNo, In_iLoopCount] := LREAL_TO_REAL(((In_lrHubG  * paarCamTable^[GVL_ConstantsFlexProfile.iCAM20_GIG, In_iLoopCount] / 100.0) +
           	(In_lrHubRG* paarCamTable^[iBewegGesetzSeg, In_iLoopCount] / 100.0 )) / (In_lrHubG  + In_lrHubRG) * 100.0) ;
				
	In_padiCam^[In_iLoopCount]:= REAL_TO_DINT(paarCamTable^[In_iCamNo, In_iLoopCount] * 1000000);
	paarTabArray^[In_iLoopCount, In_iCamNo]    := paarCamTable^[In_iCamNo, In_iLoopCount];	//Wert in "Tab_Array" (Kurvenscheibe-Punkte-Tabelle) ablegen
END_IF

END_FUNCTION

// GeneralFunctions/ILG_Functions/F_InitArray
FUNCTION F_InitArray
(* Notes on the function *)
(* Block is used to initialise arrays with an initialisation value ‘uiInitwert_in ’type UINT.							  *)
(* The array range to be initialised is parameterised as UINT: uiNo_first_array_element_in and uiNo_last_array_element_in *)
VAR_INPUT
	IN_bEnable						: BOOL;						(* input: enable *)
	IN_puiWord 						: POINTER TO WORD;  		(* input: Pointer to word *)
	IN_uiNoFirstArrayElement		: UINT;						(* input: No. of the first array element. Attention: If array goes from 62000...63999, then the first array element is [62000] and has the number "0" *)
	IN_uiNoLastArrayElement			: UINT;						(* input: No. of the last array element. Attention: If array goes from 62000...63999, then the last array element is [63999] and has the number  "1999" *)
	IN_uiInitValue					: UINT;						(* input: Init value which should be set in the range between first and last array element *)	
END_VAR
VAR
	uiLocalArrayElement 			: UINT;						(* Local counter variabel for the array element. The array element starts with "0"! *)	
END_VAR

IF IN_bEnable THEN

	//Pointer auf Startadresse setzen
	IN_puiWord := IN_puiWord + (IN_uiNoFirstArrayElement * SIZEOF(IN_puiWord^));

	FOR uiLocalArrayElement := IN_uiNoFirstArrayElement TO IN_uiNoLastArrayElement DO
		(* Wenn die Zählvariable für die Arrayelement-Nummer im Bereich des zu beschreibenden Bereichs liegt, dann beschreiben starten *)
		IN_puiWord^ := IN_uiInitValue;
		
		(* Zeiger darf erst mit dem Arrayelement Nummer 1 erhöht werden; Ein Array startet mit Nummer 0 *)
		(* 	Bitte beachten: Ein Pointer wird byte-weise hochgezählt! 
		Über die Anweisung p=p+SIZEOF(p^); kann ein Hochzählen wie im C-Compiler erreicht werden. *)
		IN_puiWord := IN_puiWord + SIZEOF(IN_puiWord^);
	END_FOR

END_IF

END_FUNCTION

// GeneralFunctions/Math/F_lrRoundRealToLReal
{attribute 'qualified_only' := ''}
{attribute 'namespace' := 'ILGStdLib.Functions.Math'}
FUNCTION F_lrRoundRealToLReal : LREAL
VAR_INPUT
	In_rValue: REAL;
	In_iDigits: INT;
END_VAR
VAR
	diValueTrunc: DINT;
	lrValueRest: LREAL;
	lrValueTemp1: LREAL;
END_VAR

lrValueTemp1:=In_rValue * EXPT(10,In_iDigits);

diValueTrunc := TRUNC_INT(lrValueTemp1);
lrValueRest := lrValueTemp1 - DINT_TO_LREAL(diValueTrunc);

IF lrValueRest < 0.5 THEN
	lrValueTemp1 := DINT_TO_LREAL(diValueTrunc) / EXPT(10,In_iDigits);
ELSE
	lrValueTemp1 := DINT_TO_LREAL(diValueTrunc+1) / EXPT(10,In_iDigits);
END_IF

F_lrRoundRealToLReal := ((TRUNC_INT(lrValueTemp1* EXPT(10,In_iDigits)))/ EXPT(10,In_iDigits));

END_FUNCTION

// GeneralFunctions/Math/F_rModulo
{attribute 'qualified_only' := ''}
{attribute 'namespace' := 'ILGStdLib.Functions.Math'}
FUNCTION F_rModulo : REAL
VAR_INPUT
	In_rValue: REAL;
	In_rModulo: REAL;
END_VAR

IF (In_rModulo = 0) THEN
	F_rModulo := In_rValue;
	RETURN;
END_IF

IF (In_rValue < 0) THEN
	F_rModulo := In_rValue;
	IF (In_rModulo > 0) THEN
		REPEAT
			F_rModulo := F_rModulo + In_rModulo ;
		UNTIL (F_rModulo >= 0)
		END_REPEAT
		RETURN;		
	ELSIF (In_rModulo < 0) THEN
		REPEAT
			F_rModulo := F_rModulo - In_rModulo ;
		UNTIL (F_rModulo >= 0)
		END_REPEAT
		F_rModulo := F_rModulo + In_rModulo ;
		RETURN;	
	END_IF 
ELSIF (In_rValue > In_rModulo) THEN
	F_rModulo := In_rValue;
	IF (In_rModulo > 0) THEN
		REPEAT
			F_rModulo := F_rModulo - In_rModulo;
		UNTIL (F_rModulo <= In_rModulo )
		END_REPEAT
		RETURN;
	ELSIF (In_rModulo < 0) THEN
		REPEAT
			F_rModulo := F_rModulo + In_rModulo;
		UNTIL (F_rModulo <= In_rModulo )
		END_REPEAT
		RETURN;
	END_IF	

ELSE F_rModulo := In_rValue;
	RETURN;
END_IF

END_FUNCTION

// GeneralFunctions/Math/F_rRound
{attribute 'qualified_only' := ''}
{attribute 'namespace' := 'ILGStdLib.Functions.Math'}
FUNCTION F_rRound : REAL
VAR_INPUT
	In_rValue: REAL;
	In_iDigits: INT;
END_VAR
VAR
	diValueTrunc: DINT;
	rValueRest: REAL;
	rValueTemp: REAL;
END_VAR

rValueTemp:=LREAL_TO_REAL(In_rValue * EXPT(10,In_iDigits));

diValueTrunc := TRUNC_INT(rValueTemp);
rValueRest := rValueTemp - DINT_TO_REAL(diValueTrunc);

IF rValueRest < 0.5 THEN
	F_rRound := DINT_TO_REAL(diValueTrunc) / LREAL_TO_REAL(EXPT(10,In_iDigits));
ELSE
	F_rRound := DINT_TO_REAL(diValueTrunc+1) / LREAL_TO_REAL(EXPT(10,In_iDigits));
END_IF

END_FUNCTION

// GeneralFunctions/Math/F_rRoundGreater
{attribute 'qualified_only' := ''}
{attribute 'namespace' := 'ILGStdLib.Functions.Math'}
FUNCTION F_rRoundGreater : REAL
VAR_INPUT
	In_rValue: REAL;
	In_iDigits: INT;
END_VAR
VAR
	diValueTrunc: DINT;
	rValueRest: REAL;
	rValueTemp: REAL;
END_VAR

rValueTemp:=In_rValue * LREAL_TO_REAL(EXPT(10,In_iDigits));

diValueTrunc := TRUNC_INT(rValueTemp);
rValueRest := rValueTemp - DINT_TO_REAL(diValueTrunc);

IF rValueRest <> 0.0 THEN
	F_rRoundGreater := DINT_TO_REAL(diValueTrunc+1) / LREAL_TO_REAL(EXPT(10,In_iDigits));
ELSE
	F_rRoundGreater := DINT_TO_REAL(diValueTrunc) / LREAL_TO_REAL(EXPT(10,In_iDigits));
END_IF

END_FUNCTION

// GeneralFunctions/Math/F_rRoundTime
{attribute 'qualified_only' := ''}
{attribute 'namespace' := 'ILGStdLib.Functions.Math'}
FUNCTION F_rRoundTime : REAL
VAR_INPUT
	In_rValue: REAL;
	In_iDigits: INT;
END_VAR
VAR
	diValueTrunc: DINT;
	rValueRest: REAL;
	rValueTemp: REAL;
END_VAR

rValueTemp:= LREAL_TO_REAL(In_rValue * EXPT(10,In_iDigits));

diValueTrunc := TRUNC_INT(rValueTemp);
rValueRest := rValueTemp - DINT_TO_REAL(diValueTrunc);

IF rValueRest < 0.5 THEN
	F_rRoundTime := DINT_TO_REAL(diValueTrunc) / LREAL_TO_REAL(EXPT(10,In_iDigits));
ELSE
	F_rRoundTime := DINT_TO_REAL(diValueTrunc+1) / LREAL_TO_REAL(EXPT(10,In_iDigits));
END_IF

IF F_rRoundTime = 0.0 THEN
	F_rRoundTime := 1.0 * LREAL_TO_REAL(EXPT(10,(-1)*In_iDigits));
END_IF

END_FUNCTION
